{region '#Template'}
	{attribute 'Version' := '5.0.0.0'}
	{attribute 'Tags' := '"LCID": "1031", "Text": "Universal, Object, BV"'}
	{attribute 'Tags' := '"LCID": "1033", "Text": "Universal, Object, BV"'}
	{attribute 'Using' := '"Type": "Template", "URI": "EC_ID"'}
	{attribute 'Using' := '"Type": "Template", "URI": "BA2_Param"'}
	{attribute 'Description' := '"LCID": "1031", "Text": "BV Wahlschalter"'}
	{attribute 'Description' := '"LCID": "1033", "Text": "BV Switch"'}
{endregion}	 
FUNCTION_BLOCK FB_BA_BV_Op_Val EXTENDS FB_BA_View
VAR_OUTPUT
	bPresentValue		: BOOL;
END_VAR
VAR_INPUT CONSTANT
	Val					: FB_BA_BV_Op;									
END_VAR

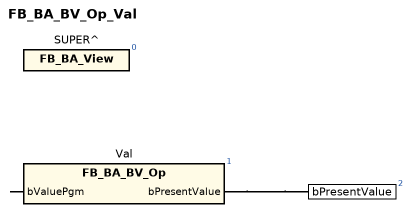
SUPER^(); // FB_BA_View
Val(); // FB_BA_BV_Op
bPresentValue := Val.bPresentValue;

METHOD FB_init : BOOL
VAR_INPUT
	bInitRetains : BOOL; // if TRUE, the retain variables are initialized (warm start / cold start)
	bInCopyCode : BOOL;  // if TRUE, the instance afterwards gets moved into the copy code (online change)
END_VAR
Val.iParent						:= THIS^;		
Val.iLabel						:= LblFun_Button; 
Val.sActiveText					:= txtEvent_On;
Val.sInactiveText				:= txtEvent_Off;
Val.bValueRm					:= FALSE;
Val.eToggleMode 				:= E_BA_ToggleMode.eSwitch;
END_METHOD

END_FUNCTION_BLOCK

(* stored: Version 1.1.0.1, ProductVersion 3.1.4024.12
   POU FB_BA_BV_Op_Val: Id {6f467657-a6b6-43c5-a9df-f79eaac24583}, SpecialFunc None
   Method FB_init: Id {8507c858-a193-4ec7-ae08-8718b91f6e31} *)
